// instrumetn kinematic paramters
TYPE ST_InstruKinematicParam :
STRUCT	
	
	// instrument geometric parameters
	// NOTE: need update based on instrument types
	m_rodLength:LREAL:=0.5392;
	m_headLength:LREAL :=0.01;
	m_fingerLength:LREAL :=0;
	m_maxGripAngle :LREAL := 50.0 * g_deg2Rad;
	m_minGripAngle :LREAL := -25 * g_deg2Rad; // make sure fingers are fully closed
	
	// instrument kinematic parameters for joint/DH space transformation
	kx:lreal:=1;
	ky:lreal:=1;
	kz:LREAL:=1;
	k13:LREAL:=0.775;
	k23:LREAL:=0.775;
	m_openAngleDir:INT:=-1;
	
	// instrument wrist DH joint limit
	m_wristMinDHJntPos :Vec3d;
	m_wristMaxDHJntPos :Vec3d;

END_STRUCT
END_TYPE

(* stored: Version 1.1.0.1, ProductVersion 3.1.4024.12
   DUT ST_InstruKinematicParam: Id {c902676e-88fd-4523-9f32-42df361ddc7d} *)
